Universal Robots PolyScope program: gripper_tutorial2.urp

Program gripper_tutorial2 (installation=default directory=/programs/usbdisk_0 createdIn=3.3.0.0 lastSavedIn=3.10.1.76190 robotSerialNumber=2017356443)
Calibrated DH parameters: a=[0.000092, -0.116521, -0.182101, -0.000106, 0.000044, 0]; d=[0.089391, 255.189113, -82.629387, -172.449369, 0.094782, 0.082637]; alpha=[1.569598, 0.001603, 0.002015, 1.570234, -1.570307, 0]; deltaTheta=[-0.000017, 1.293309, -0.204843, -1.088417, 0.000036, -0.000078]
Robot Program (runOnlyOnce=true)
  Popup Warning (haltProgram=false message=Don't modify this program. It will be erased at next boot. inputType=Text)
  'Activate the gripper before controling it'
  Popup Message (haltProgram=false message=Activate the gripper before controling it inputType=Text)
  Script: rq_activate_and_wait()
  'Fully close the gripper and wait for completion'
  Popup Message (haltProgram=false message=Fully close the gripper and wait for completion inputType=Text)
  URCap Gripper (Robotiq_2-Finger_Adaptive_Gripper, Robotiq Inc.) dataModel(position=100, force=100, speed=79, blocking=true)
  'Fully open the gripper and wait for completion'
  Popup Message (haltProgram=false message=Fully open the gripper and wait for completion inputType=Text)
  URCap Gripper (Robotiq_2-Finger_Adaptive_Gripper, Robotiq Inc.) dataModel(position=0, force=100, speed=79, blocking=true)
  'Partially close the gripper and wait for completion'
  Popup Message (haltProgram=false message=Partially close the gripper and wait for completion inputType=Text)
  URCap Gripper (Robotiq_2-Finger_Adaptive_Gripper, Robotiq Inc.) dataModel(position=31, force=100, speed=79, blocking=true)
  'Close the gripper and test the object detection'
  Popup Message (haltProgram=false message=Close the gripper and test the object detection inputType=Text)
  URCap Gripper (Robotiq_2-Finger_Adaptive_Gripper, Robotiq Inc.) dataModel(position=100, force=100, speed=79, blocking=true)
  If rq_is_object_detected()
    'An object has been detected'
    Popup Message (haltProgram=false message=An object has been detected inputType=Text)
  Else 
    'No object detected'
    Popup Message (haltProgram=false message=No object detected inputType=Text)
  'Get the gripper current position in %. 100% is reached when the grippers is in encompassing mode.'
  Script: popup(rq_get_position(), "Gripper position (%)", blocking=True)
  'Command the gripper to open and continue the program execution.'
  Popup Message (haltProgram=false message=Command the gripper to open and continue the program execution. inputType=Text)
  URCap Gripper (Robotiq_2-Finger_Adaptive_Gripper, Robotiq Inc.) dataModel(position=0, force=0, speed=0, blocking=false)
  'You can insert robot movement instructions while the gripper is moving'
  Wait Condition expression=rq_is_motion_complete()
  'Gripper motion completed'
  Popup Message (haltProgram=false message=Gripper motion completed inputType=Text)
  Folder Script Funtions
    Halt
    Folder Functions operating on a 0-100 span
      'Sets the gripper force [0-100]'
      Script: rq_set_force_norm(50)
      'Sets the gripper speed [0-100]'
      Script: rq_set_speed_norm(75)
      'Sends the partial move command and continue [0-100]'
      Script: rq_move_norm(75)
      'Sends the partial move command and wait until completion. [0-100]'
      Script: rq_move_and_wait_norm(30)
      'Sets the target position [0-100]'
      Script: rq_set_pos_norm(45)
      'Returns the gripper current position [0-100]'
      position := rq_current_pos_norm()
    Folder Functions operating on a 0-255 span
      'Sends the partial move command and wait until completion. [0-255]'
      Script: rq_move_and_wait(150)
      'Sets the target position'
      Script: rq_set_pos(150)
      'Returns the gripper current position [0-255]'
      position := rq_current_pos()
      'Sends the partial move command and continue'
      Script: rq_move(150)
      'Sets the gripper speed [0-255]'
      Script: rq_set_speed(255)
      'Sets the gripper force [0-255]'
      Script: rq_set_force(255)
    Folder Functions independant of the span
      'Activate the gripper if needed and wait for completion'
      Script: rq_activate_and_wait()
      'Activate the gripper and continue execution'
      Script: rq_activate()
      'Wait the end of activation'
      Wait Condition expression=rq_is_gripper_activated()
      'Sends the open command and continue'
      Script: rq_open()
      'Send the close command and continue'
      Script: rq_close()
      'Returns True if the motion is completed.'
      motion_complete := rq_is_motion_complete()
      'Returns True if an object has been detected.'
      object_detected := rq_is_object_detected()
      'Sends the open command and wait until completion'
      Script: rq_open_and_wait()
      'Sends the close command and wait until completion'
      Script: rq_close_and_wait()
      'Sets the goto bit to 1. Refer to user manual.'
      Script: rq_go_to()
      'Stops motion. The goto bit is cleared.'
      Script: rq_stop()
      'Sends the closing autorelease instruction and wait until completion'
      Script: rq_auto_release_close_and_wait()
      'Sends the opening autorelease instruction and wait until completion'
      Script: rq_auto_release_open_and_wait()
      'Resets the activation status of the gripper. Use after an autorelease before activating the gripper.'
      Script: rq_reset()
